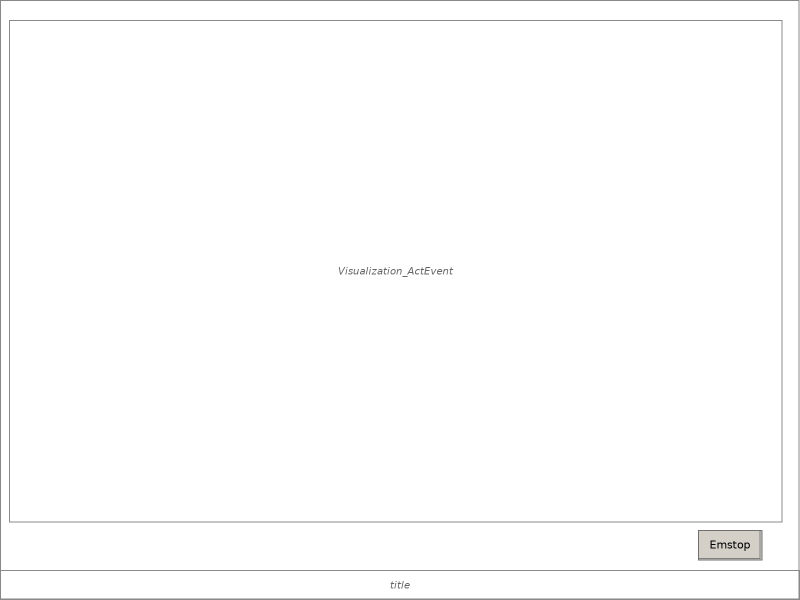
VISUALIZATION vis_arm  // 800x600
    Frame (0,570 800x30)
        shows title()
    TabControl (9,20 773x502)
        shows Visualization_ActEvent()
        shows Visualization_LogEvent()
        shows Vis101()
        [0]: TabTitle=ActEvent
        [1]: TabTitle=LogEvent
    Button (698,530 64x30), "Emstop", colour toggle: GVL.HMI_btEmstop
        toggle GVL.HMI_btEmstop
END_VISUALIZATION

(* stored: Version 1.1.0.1, ProductVersion 3.1.4024.11
   Visu vis_arm: Id {500c6321-ac7a-4d11-8e94-75d7f742b380} *)
